PROGRAM PRG_TESTS
VAR
    // We declare instances of our test suites here
    DigitalSensorTest : FB_DigitalSensor_Test;
    
    // NEW: Add the Main Machine test suite
    MainMachineTest   : FB_MainMachine_Test; 
END_VAR

// This is the master command that tells TcUnit to run all tests and print the results
TcUnit.RUN();

END_PROGRAM

(* stored: Version 1.1.0.1
   POU PRG_TESTS: Id {41a4f515-a6f7-46c3-a9c6-f5a4d8f8a294}, SpecialFunc None *)
